FUNCTION_BLOCK AppContext EXTENDS TcoCore.TcoContext
VAR
	_station001 : Station001(THIS^);
END_VAR

(*~
	<docu>
		<summary>
			Main method of the TcoContext. This is the entry point of any control logic that belongs to this context. 
			The call of this method is ensured by calling the <c>InstanceName.Run()</c> method, and it must not be called explicitly.
			This method is abstract, and it must be overridden in derived block.
		</summary>
	</docu>
~*)
METHOD PROTECTED  Main
_station001();
END_METHOD

END_FUNCTION_BLOCK

(* stored: Version 1.1.0.1, ProductVersion 3.1.4024.9
   POU AppContext: Id {e82506b0-90bc-42b7-916c-c4162fa94076}, SpecialFunc None
   Method Main: Id {a771a6c3-fdd4-4888-9f96-785131531d33} *)
